FUNCTION_BLOCK TriggerPoint IMPLEMENTS I_Cyclic, I_Resettable, I_Object
VAR
	_TriggerPointMovers : ARRAY[0..MaxMovers] OF I_XtsMover;
	SystemMovers : ARRAY[0..MaxMovers] OF I_XtsMover;
	NumberOfMovers : INT;
	_position : LREAL;
	_range : LREAL;
END_VAR
VAR CONSTANT
	MaxMovers : INT := 10;
END_VAR

METHOD Cycle : HRESULT
VAR 
	i : INT;
	arrivingMover : I_XtsMover;
	detected : BOOL;
END_VAR
FOR i := 0 TO MaxMovers DO
	IF SystemMovers[i] <> 0 THEN
		IF SystemMovers[i].AxisRef.NcToPlc.ModuloActPos < _position + 10.0 AND
			SystemMovers[i].AxisRef.NcToPlc.ModuloActPos > _position - 10.0 THEN
			arrivingMover := SystemMovers[i];
		END_IF
	END_IF
END_FOR
IF arrivingMover <> 0 THEN
	FOR i := 0 TO MaxMovers DO
		IF arrivingMover = _TriggerPointMovers[i] THEN
			detected := TRUE;
		END_IF
	END_FOR
	IF NOT detected THEN
		FOR i := 0 TO MaxMovers DO
			IF _TriggerPointMovers[i] = 0 THEN
				_TriggerPointMovers[i] := arrivingMover;
				EXIT;
			END_IF
		END_FOR
	END_IF
END_IF
FOR i := 0 TO MaxMovers DO
	IF _TriggerPointMovers[i] <> 0 AND_THEN 
		_TriggerPointMovers[i].AxisRef.NcToPlc.ModuloActPos > _position + _range THEN
		_TriggerPointMovers[i] := 0;
	END_IF
END_FOR
END_METHOD

//FB_Init is always available implicitly and it is used primarily for initialization.
//The return value is not evaluated. For a specific influence, you can also declare the
//methods explicitly and provide additional code there with the standard initialization
//code. You can evaluate the return value.
METHOD FB_Init: BOOL
VAR_INPUT
    bInitRetains: BOOL; // TRUE: the retain variables are initialized (reset warm / reset cold)
    bInCopyCode: BOOL;  // TRUE: the instance will be copied to the copy code afterward (online change)   
	Position : LREAL;
	Range : LREAL;
END_VAR
_range := Range;
_position := Position;
END_METHOD

PROPERTY Position : lreal
GET
Position := _Position;
END_GET
END_PROPERTY

METHOD RegisterMovers : HRESULT
VAR_INPUT
	MyMover : I_XtsMover;
END_VAR
VAR
	i : uINT;
END_VAR
IF MyMover <> 0 THEN
	SystemMovers[NumberOfMovers] := MyMover;
	NumberOfMovers := NumberOfMovers + 1;
ELSE
	RegisterMovers := -1;
END_IF
END_METHOD

METHOD RegisterWithParent
VAR_INPUT
	Parent	: Base_Library.I_HostObjects;
END_VAR
END_METHOD

METHOD Reset : HRESULT
VAR
	i : INT;
END_VAR
FOR i := 0 TO MaxMovers DO
	_TriggerPointMovers[i] := 0;
END_FOR
END_METHOD

END_FUNCTION_BLOCK

(* stored: Version 1.1.0.1
   POU TriggerPoint: Id {3b207e24-d75e-4621-b3ed-6508fa0edd6b}, SpecialFunc None
   Method Cycle: Id {d6eab57b-cfae-4645-975e-c4c454010bba}
   Method FB_Init: Id {e845fedb-d2ed-4b96-bd3d-fedfbc78ddd6}
   Property Position: Id {c71cd478-609b-4fc2-8d05-30d780bf9546}
   Get Get: Id {451cf0fe-6fca-4a29-afbe-d1677f0ae1dd}
   Method RegisterMovers: Id {44c86865-f914-40c8-9d7f-ebabcc61d481}
   Method RegisterWithParent: Id {37f95e6a-9c59-4bc9-8631-6fedca7eef6e}
   Method Reset: Id {8a4824d9-717e-48ab-a44e-c26909b89697} *)
